// SIMATIC S7-200 project (STEP 7-Micro/WIN), CPU 224XP REL 02.01

ORGANIZATION_BLOCK 主程序:OB1
TITLE=程序注释
BEGIN
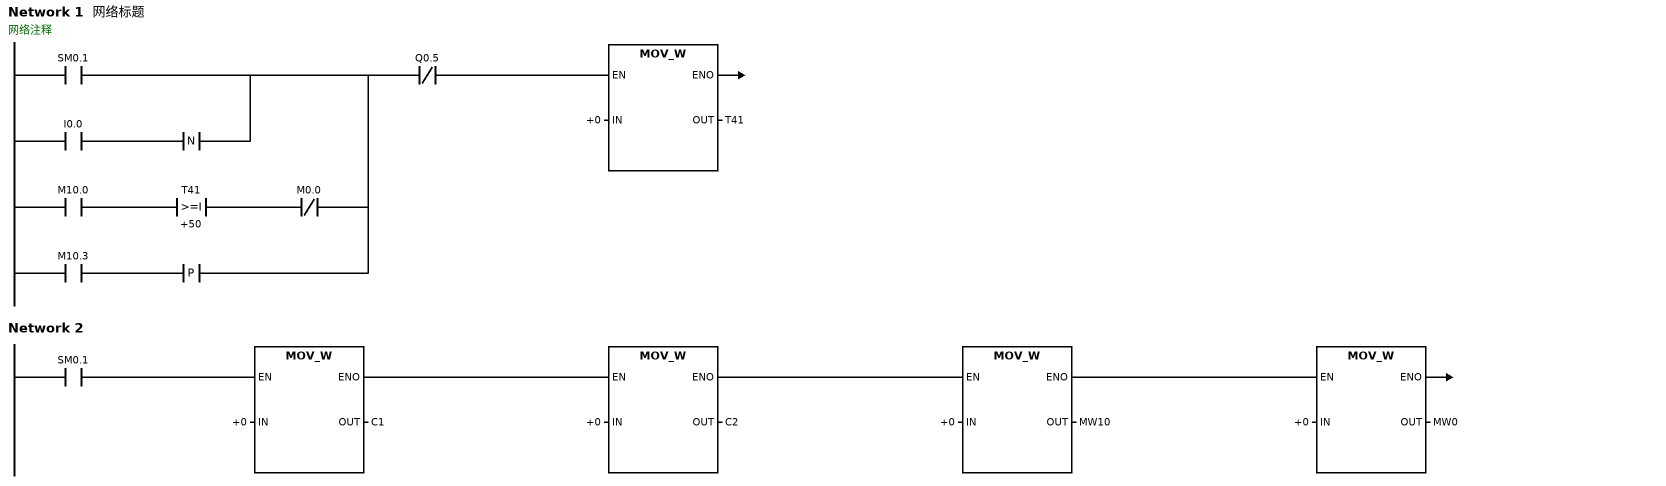
Network 1 // 网络标题
// 网络注释
LD     SM0.1
LD     I0.0
ED
OLD
LD     M10.0
AW>=   T41, +50
AN     M0.0
OLD
LD     M10.3
EU
OLD
AN     Q0.5
MOVW   +0, T41
Network 2
LD     SM0.1
MOVW   +0, C1
AENO
MOVW   +0, C2
AENO
MOVW   +0, MW10
AENO
MOVW   +0, MW0
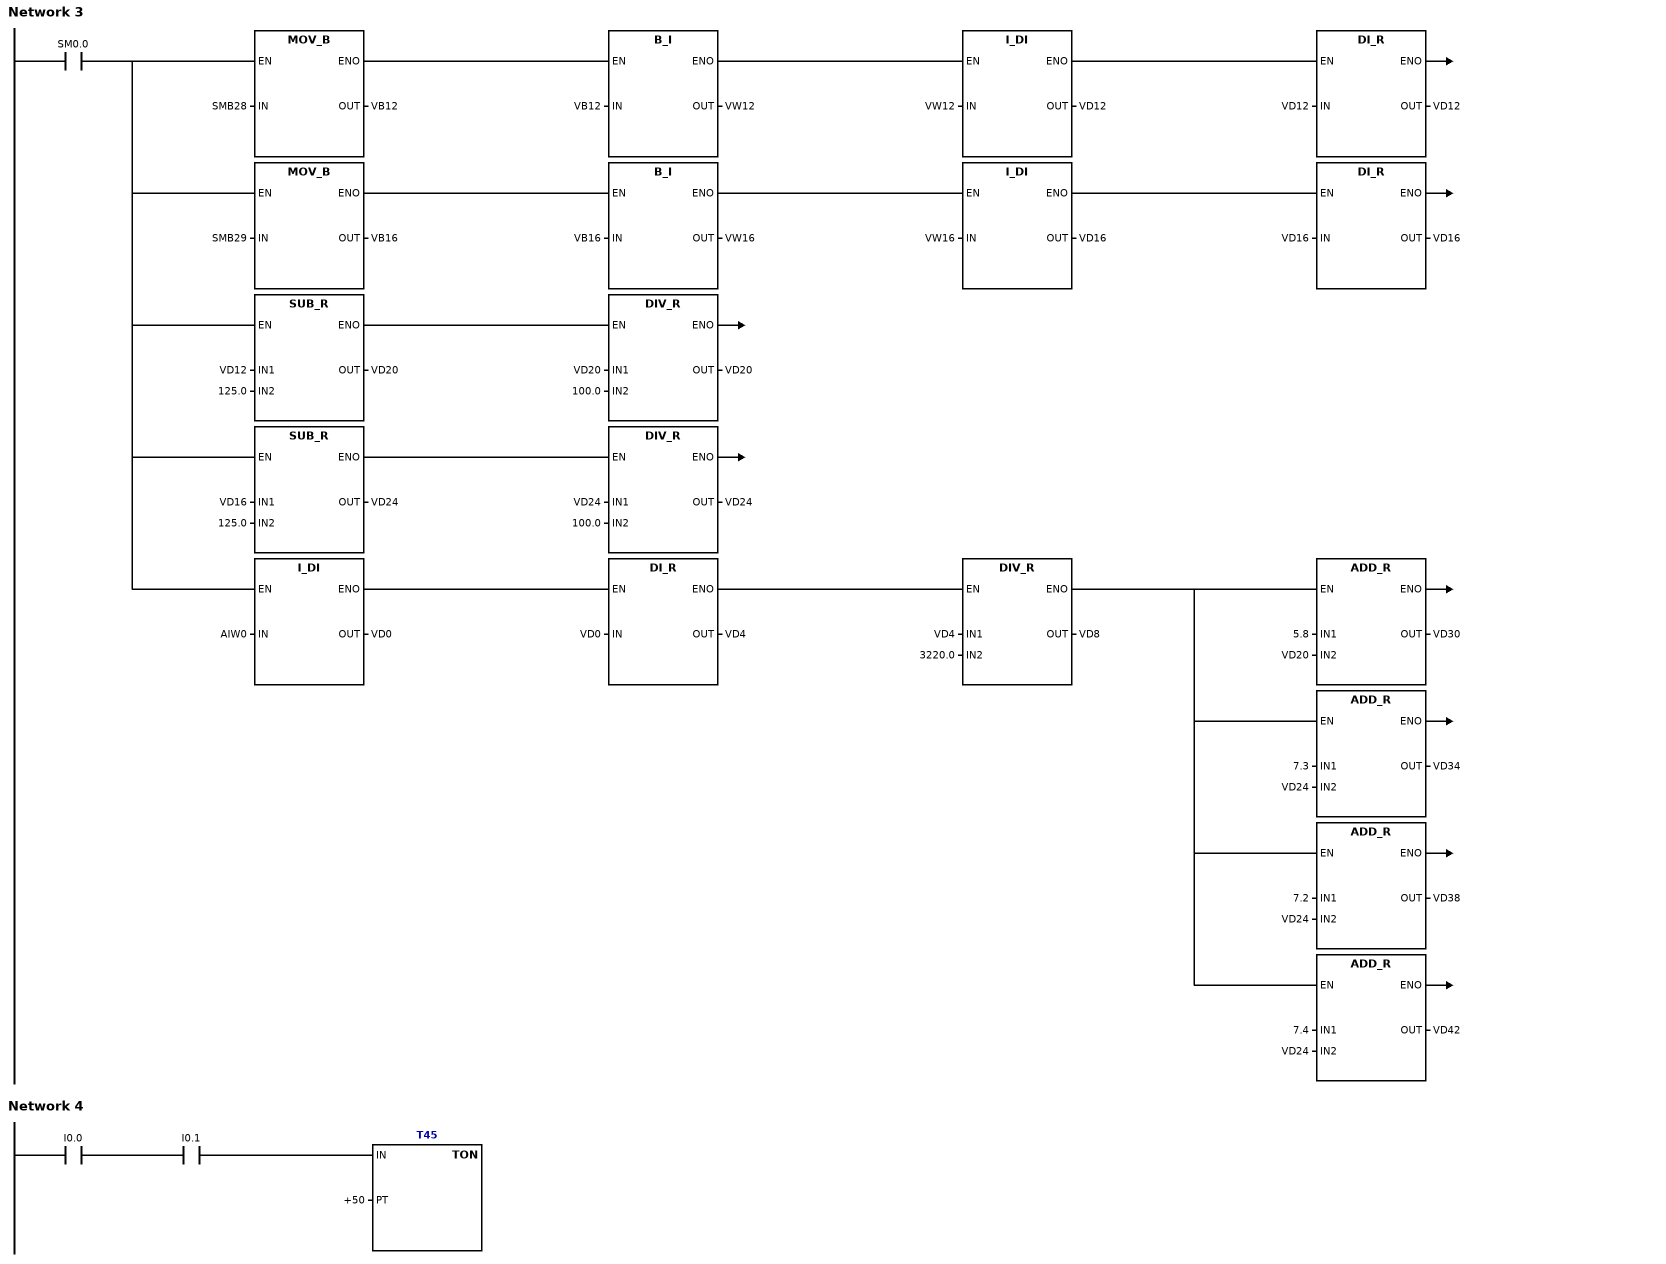
Network 3
LD     SM0.0
LPS
MOVB   SMB28, VB12
AENO
BTI    VB12, VW12
AENO
ITD    VW12, VD12
AENO
DTR    VD12, VD12
LRD
MOVB   SMB29, VB16
AENO
BTI    VB16, VW16
AENO
ITD    VW16, VD16
AENO
DTR    VD16, VD16
LRD
MOVR   VD12, VD20
AENO
-R     125.0, VD20
AENO
/R     100.0, VD20
LRD
MOVR   VD16, VD24
AENO
-R     125.0, VD24
AENO
/R     100.0, VD24
LPP
ITD    AIW0, VD0
AENO
DTR    VD0, VD4
AENO
MOVR   VD4, VD8
AENO
/R     3220.0, VD8
AENO
MOVR   5.8, VD30
+R     VD20, VD30
MOVR   7.3, VD34
+R     VD24, VD34
MOVR   7.2, VD38
+R     VD24, VD38
MOVR   7.4, VD42
+R     VD24, VD42
Network 4
LD     I0.0
A      I0.1
TON    T45, +50
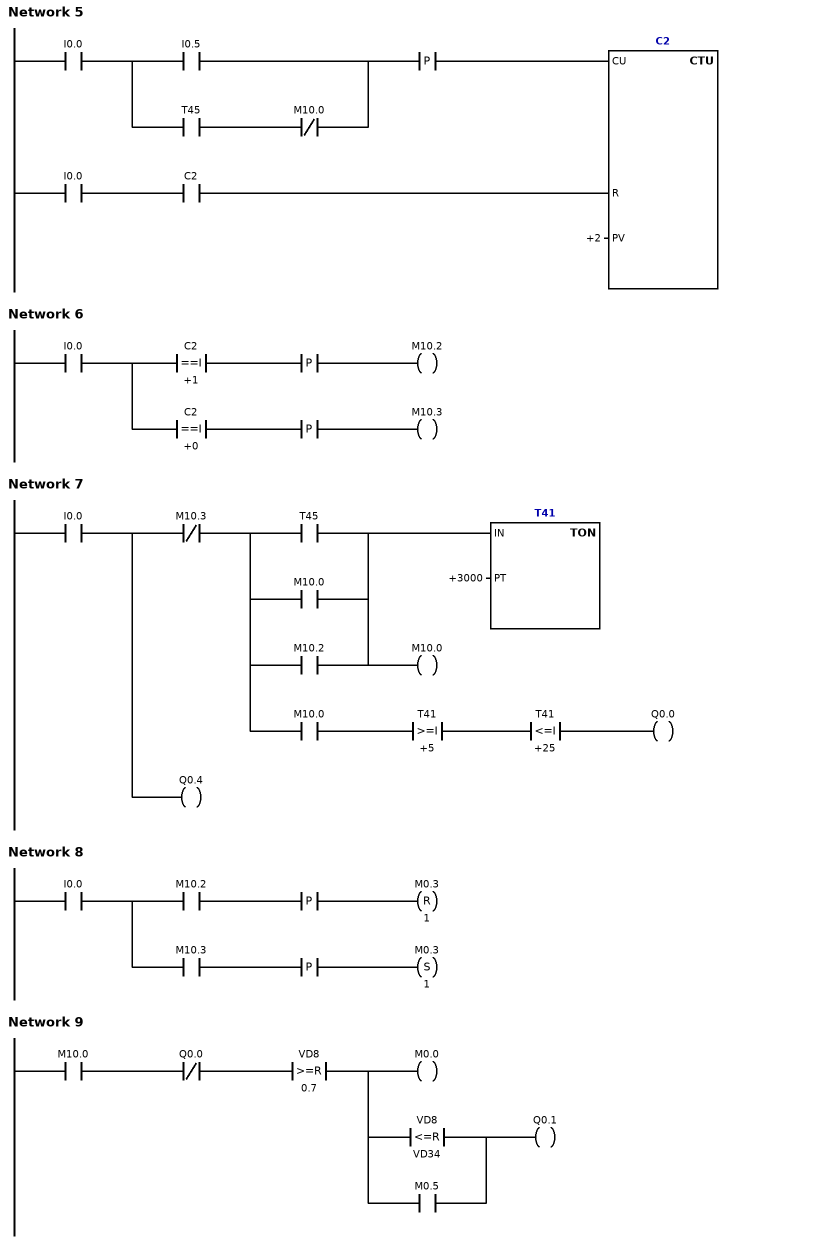
Network 5
LD     I0.0
LD     I0.5
LD     T45
AN     M10.0
OLD
ALD
EU
LD     I0.0
A      C2
CTU    C2, +2
Network 6
LD     I0.0
LPS
AW=    C2, +1
EU
=      M10.2
LPP
AW=    C2, +0
EU
=      M10.3
Network 7
LD     I0.0
LPS
AN     M10.3
LPS
LD     T45
O      M10.0
O      M10.2
ALD
TON    T41, +3000
=      M10.0
LPP
A      M10.0
AW>=   T41, +5
AW<=   T41, +25
=      Q0.0
LPP
=      Q0.4
Network 8
LD     I0.0
LPS
A      M10.2
EU
R      M0.3, 1
LPP
A      M10.3
EU
S      M0.3, 1
Network 9
LD     M10.0
AN     Q0.0
AR>=   VD8, 0.7
=      M0.0
LDR<=  VD8, VD34
O      M0.5
ALD
=      Q0.1
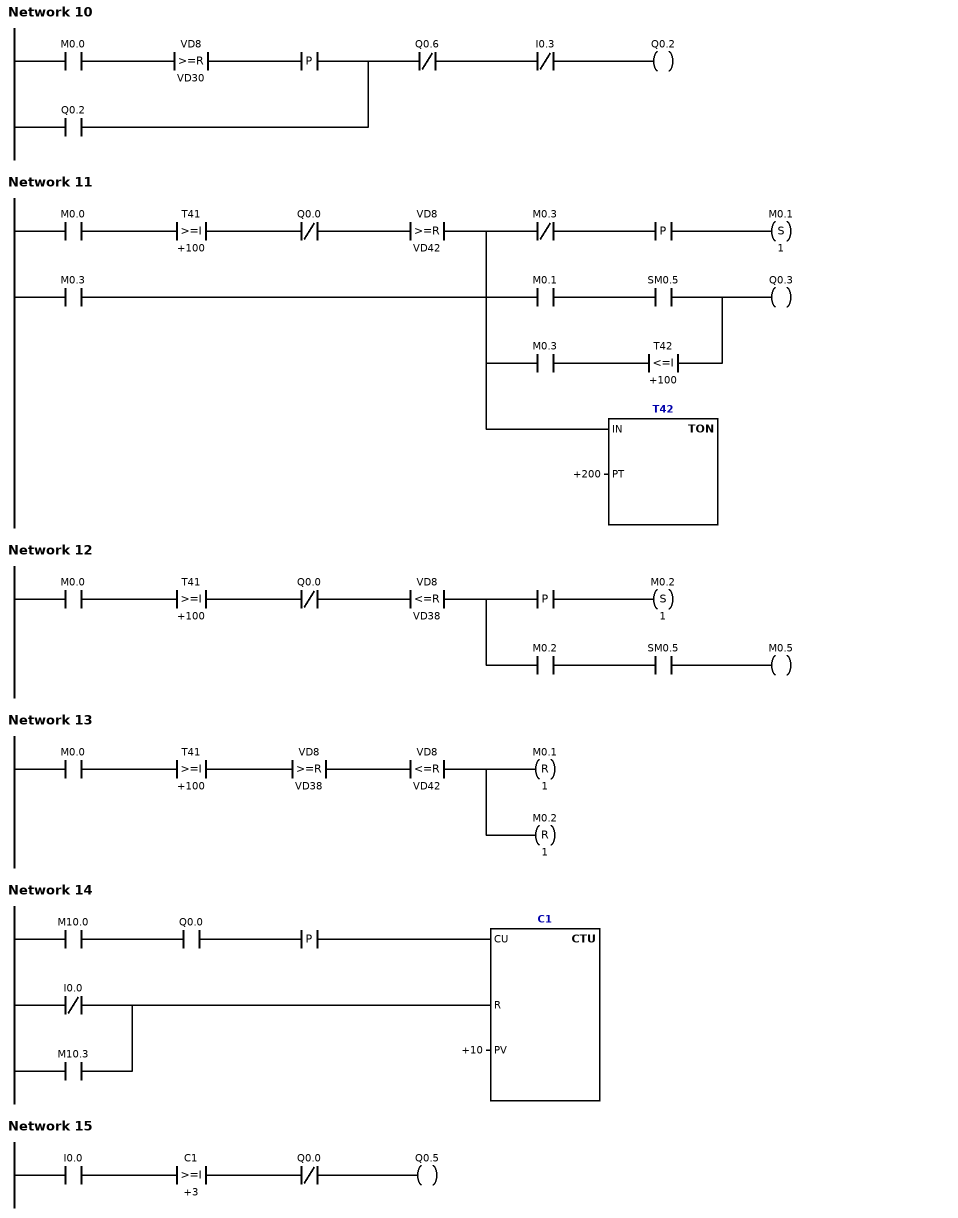
Network 10
LD     M0.0
AR>=   VD8, VD30
EU
O      Q0.2
AN     Q0.6
AN     I0.3
=      Q0.2
Network 11
LD     M0.0
AW>=   T41, +100
AN     Q0.0
AR>=   VD8, VD42
O      M0.3
LPS
AN     M0.3
EU
S      M0.1, 1
LRD
LD     M0.1
A      SM0.5
LD     M0.3
AW<=   T42, +100
OLD
ALD
=      Q0.3
LPP
TON    T42, +200
Network 12
LD     M0.0
AW>=   T41, +100
AN     Q0.0
AR<=   VD8, VD38
LPS
EU
S      M0.2, 1
LPP
A      M0.2
A      SM0.5
=      M0.5
Network 13
LD     M0.0
AW>=   T41, +100
AR>=   VD8, VD38
AR<=   VD8, VD42
R      M0.1, 1
R      M0.2, 1
Network 14
LD     M10.0
A      Q0.0
EU
LDN    I0.0
O      M10.3
CTU    C1, +10
Network 15
LD     I0.0
AW>=   C1, +3
AN     Q0.0
=      Q0.5
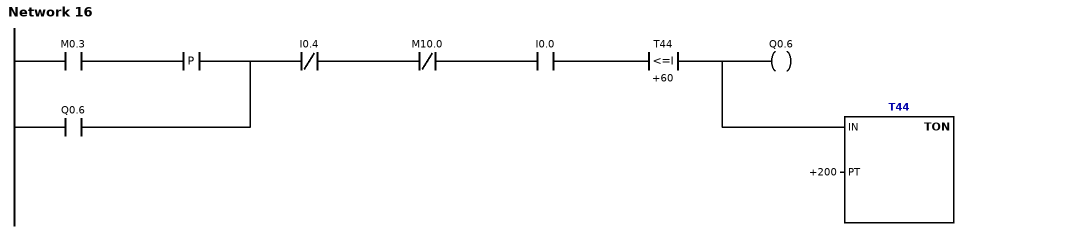
Network 16
LD     M0.3
EU
O      Q0.6
AN     I0.4
AN     M10.0
A      I0.0
AW<=   T44, +60
=      Q0.6
TON    T44, +200
END_ORGANIZATION_BLOCK
